FUNCTION_BLOCK SET_AT_INDEX
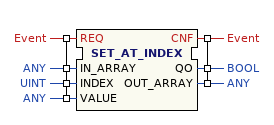
  EVENT_INPUT
    REQ WITH IN_ARRAY, INDEX, VALUE;
  END_EVENT
  EVENT_OUTPUT
    CNF WITH QO, OUT_ARRAY;
  END_EVENT
  VAR_INPUT
    IN_ARRAY : ANY;
    INDEX : UINT;
    VALUE : ANY;
  END_VAR
  VAR_OUTPUT
    QO : BOOL;
    OUT_ARRAY : ANY;
  END_VAR
END_FUNCTION_BLOCK
